// TIA Portal V19 export
FUNCTION "Route 405" : Void   // FC104, STL
TITLE = Polygon Transfer Line - SIP Sequence
{ S7_Optimized_Access := 'TRUE' }
// stored: AutoNumber false
   VAR_TEMP
      device_fault : Bool;
      switch_fault : Bool;
      tmp : Bool;
      Step_on : Bool;
      Dev_Check : Bool;
      New_Msg : Bool;
      Route_Ready : Bool;   // Ready to Run
      PNIOnodeFault : Bool;
      StepTime : S5Time;
      TimerError : Int;
      scratch_DI : DInt;
      scratch_Real : Real;
      Message : Int;
      scratch_I : Int;
      tmpWord : Word;
      PNIODiag : Struct
         node_2 : Struct
            failed : Bool;
            moduleFault : Bool;
         END_STRUCT;
         node_3 : Struct
            failed : Bool;
            moduleFault : Bool;
         END_STRUCT;
         node_4 : Struct
            failed : Bool;
            moduleFault : Bool;
         END_STRUCT;
         node_5 : Struct
            failed : Bool;
            moduleFault : Bool;
         END_STRUCT;
         node_6 : Struct
            failed : Bool;
            moduleFault : Bool;
         END_STRUCT;
         node_7 : Struct
            failed : Bool;
            moduleFault : Bool;
         END_STRUCT;
         node_8 : Struct
            failed : Bool;
            moduleFault : Bool;
         END_STRUCT;
         node_9 : Struct
            failed : Bool;
            moduleFault : Bool;
         END_STRUCT;
         node_10 : Struct
            failed : Bool;
            moduleFault : Bool;
         END_STRUCT;
         node_11 : Struct
            failed : Bool;
            moduleFault : Bool;
         END_STRUCT;
         node_12 : Struct
            failed : Bool;
            moduleFault : Bool;
         END_STRUCT;
      END_STRUCT;
      __PlcmigTempFillBits_38B0 : Array[0..7] of Bool;
   END_VAR
BEGIN

NETWORK
TITLE = PNIO 100 Node Faults
// PNIO Node 2
// PNIO Node 2
      A     "Module Diagnostic Result"."2_AL1103".ErrorValue.%X1;
      =     #PNIODiag.node_2.failed;
      A     "Module Diagnostic Result"."2_AL1103".ErrorValue.%X2;
      =     #PNIODiag.node_2.moduleFault;
// PNIO Node 3
      A     "Module Diagnostic Result"."3_AL1307".ErrorValue.%X1;
      =     #PNIODiag.node_3.failed;
      A     "Module Diagnostic Result"."3_AL1307".ErrorValue.%X2;
      =     #PNIODiag.node_3.moduleFault;
// PNIO Node 4
      A     "Module Diagnostic Result"."4_AL1307".ErrorValue.%X1;
      =     #PNIODiag.node_4.failed;
      A     "Module Diagnostic Result"."4_AL1307".ErrorValue.%X2;
      =     #PNIODiag.node_4.moduleFault;
// PNIO Node 5
      A     "Module Diagnostic Result"."5_AL1307".ErrorValue.%X1;
      =     #PNIODiag.node_5.failed;
      A     "Module Diagnostic Result"."5_AL1307".ErrorValue.%X2;
      =     #PNIODiag.node_5.moduleFault;
// PNIO Node 6
      A     "Module Diagnostic Result"."6_AL1307".ErrorValue.%X1;
      =     #PNIODiag.node_6.failed;
      A     "Module Diagnostic Result"."6_AL1307".ErrorValue.%X2;
      =     #PNIODiag.node_6.moduleFault;
// PNIO Node 7
      A     "Module Diagnostic Result"."7_AL1307".ErrorValue.%X1;
      =     #PNIODiag.node_7.failed;
      A     "Module Diagnostic Result"."7_AL1307".ErrorValue.%X2;
      =     #PNIODiag.node_7.moduleFault;
// PNIO Node 8
      A     "Module Diagnostic Result"."8_Promag300".ErrorValue.%X1;
      =     #PNIODiag.node_8.failed;
      A     "Module Diagnostic Result"."8_Promag300".ErrorValue.%X2;
      =     #PNIODiag.node_8.moduleFault;
// PNIO Node 9
      A     "Module Diagnostic Result"."9_SinaG120".ErrorValue.%X1;
      =     #PNIODiag.node_9.failed;
      A     "Module Diagnostic Result"."9_SinaG120".ErrorValue.%X2;
      =     #PNIODiag.node_9.moduleFault;
// PNIO Node 10
      A     "Module Diagnostic Result"."10_AL1307".ErrorValue.%X1;
      =     #PNIODiag.node_10.failed;
      A     "Module Diagnostic Result"."10_AL1307".ErrorValue.%X2;
      =     #PNIODiag.node_10.moduleFault;
// PNIO Node 11
      A     "Module Diagnostic Result"."11_PNCoup".ErrorValue.%X1;
      =     #PNIODiag.node_11.failed;
      A     "Module Diagnostic Result"."11_PNCoup".ErrorValue.%X2;
      =     #PNIODiag.node_11.moduleFault;
// PNIO Node 12
      A     "Module Diagnostic Result"."12_AL1307".ErrorValue.%X1;
      =     #PNIODiag.node_12.failed;
      A     "Module Diagnostic Result"."12_AL1307".ErrorValue.%X2;
      =     #PNIODiag.node_12.moduleFault;


NETWORK
TITLE = PNIO node fault
      O     #PNIODiag.node_2.failed;
      O     #PNIODiag.node_2.moduleFault;
      O     #PNIODiag.node_3.failed;
      O     #PNIODiag.node_3.moduleFault;
      O     #PNIODiag.node_4.failed;
      O     #PNIODiag.node_4.moduleFault;
      O     #PNIODiag.node_5.failed;
      O     #PNIODiag.node_5.moduleFault;
      O     #PNIODiag.node_6.failed;
      O     #PNIODiag.node_6.moduleFault;
      O     #PNIODiag.node_7.failed;
      O     #PNIODiag.node_7.moduleFault;
      O     #PNIODiag.node_8.failed;
      O     #PNIODiag.node_8.moduleFault;
      O     #PNIODiag.node_9.failed;
      O     #PNIODiag.node_9.moduleFault;
      O     #PNIODiag.node_10.failed;
      O     #PNIODiag.node_10.moduleFault;
      O     #PNIODiag.node_11.failed;
      O     #PNIODiag.node_11.moduleFault;
      O     #PNIODiag.node_12.failed;
      O     #PNIODiag.node_12.moduleFault;
      =     #PNIOnodeFault;


NETWORK
TITLE = Device Faults
      O     "ItemAlarmsOP".Item[20];  //FB_FAULT_VALVE_09_05
      O     "ItemAlarmsOP".Item[23];  //FB_FAULT_VALVE_09_08
      O     "ItemAlarmsOP".Item[24];  //FB_FAULT_VALVE_09_09
      O     "ItemAlarmsOP".Item[25];  //FB_FAULT_VALVE_09_10
      O     "ItemAlarmsOP".Item[26];  //FB_FAULT_VALVE_09_11
      O     "ItemInfoScada".Items[68].fb_error;
      O     "ItemInfoScada".Items[69].fb_error;
      O     "ItemInfoScada".Items[70].fb_error;
      O     "ItemInfoScada".Items[85].fb_error;
      O     "ItemInfoScada".Items[71].fb_error;
      O     "ItemInfoScada".Items[72].fb_error;
      O     "ItemInfoScada".Items[73].fb_error;
      O     "ItemInfoScada".Items[74].fb_error;
      O     "ItemInfoScada".Items[75].fb_error;
      O     "ItemInfoScada".Items[76].fb_error;
      O     "ItemInfoScada".Items[78].fb_error;
      O     "ItemInfoScada".Items[79].fb_error;
      O     "ItemInfoScada".Items[80].fb_error;
      O     "ItemInfoScada".Items[81].fb_error;
      O     "ItemInfoScada".Items[82].fb_error;
      O     "ItemInfoScada".Items[83].fb_error;
      O     "ItemInfoScada".Items[77].fb_error;
      O     "ItemInfoScada".Items[84].fb_error;
      O     "ItemInfoScada".Items[77].TrippedInd;
      O     "ItemInfoScada".Items[77].IsolatedInd;
      O     "ItemInfoScada".Items[84].TrippedInd;
      O     "ItemInfoScada".Items[84].IsolatedInd;
      O     #PNIOnodeFault;
      O     "ProcessAndPbAlarms"."A"[78];  //A78_PG_PTX0940HighPress
      AN    "RTE_405_TestBit";
      =     #device_fault;

NETWORK
TITLE = Switch Fault
      A(;
      ON    "PG_Devices".DI_100_005_X06_X1_3p4;
      O     "PG_Devices".DI_100_005_X06_X1_3p2;
      O     "PG_Devices".DI_100_012_X1_1p2;
      );
      AN    "RTE_405_TestBit";
      =     #switch_fault;

NETWORK
TITLE = Set Devices in Auto
      A     "RTE_405_DB".HMI.RUNNING;
      R     "ItemInfoScada".Items[50].auto_man;
      R     "ItemInfoScada".Items[53].auto_man;
      R     "ItemInfoScada".Items[54].auto_man;
      R     "ItemInfoScada".Items[55].auto_man;
      R     "ItemInfoScada".Items[56].auto_man;
      R     "ItemInfoScada".Items[69].auto_man;
      R     "ItemInfoScada".Items[70].auto_man;
      R     "ItemInfoScada".Items[68].auto_man;
      R     "ItemInfoScada".Items[72].auto_man;
      R     "ItemInfoScada".Items[73].auto_man;
      R     "ItemInfoScada".Items[75].auto_man;
      R     "ItemInfoScada".Items[76].auto_man;
      R     "ItemInfoScada".Items[78].auto_man;
      R     "ItemInfoScada".Items[79].auto_man;
      R     "ItemInfoScada".Items[80].auto_man;
      R     "ItemInfoScada".Items[81].auto_man;
      R     "ItemInfoScada".Items[82].auto_man;
      R     "ItemInfoScada".Items[83].auto_man;
      R     "ItemInfoScada".Items[77].auto_man;
      R     "ItemInfoScada".Items[84].auto_man;

NETWORK
TITLE = Route Healthy
      AN    #device_fault;
      AN    #switch_fault;
      =     "RTE_405_DB".HMI.Route_Healthy;

NETWORK
TITLE = DEVICE FAULT STATUS
      A     #device_fault;
      =     "RTE_405_DB".FLAGS.Device_Fault;

NETWORK
TITLE = GENERAL FAULT STATUS
      O     #switch_fault;
      O     "RTE_405_DB".FLAGS.Device_Fault;
      A     "RTE_405_DB".HMI.RUNNING;
      =     "RTE_405_DB".HMI.FAULT;

NETWORK
TITLE = Temporary Message Store
// Clear down temporary message store.
      L     0;
      T     #Message;
      NOP   0;

NETWORK
TITLE = Generate Sequence Start Command
// The sequence is initiated via the interface signals ..afl
      A     "RTE_405_DB".HMI_CMD.Start;
      AN    "RTE_405_DB".HMI.RUNNING;
      A     "RTE_405_DB".HMI.Route_Healthy;
      =     "RTE_405_DB".FLAGS.Sequence_Start;

      AN    "RTE_405_DB".HMI.RUNNING;
      A     "RTE_405_DB".HMI.Route_Healthy;
      =     "RTE_405_DB".HMI_CMD.Start_Available;


NETWORK
TITLE = ****ERROR MESSAGE****
// Message 10 - Device Fault
      A(;
      O     "RTE_405_DB".HMI_CMD.Start;
      O     "RTE_405_DB".HMI_CMD.Continue;
      );
      A     #device_fault;
      JNB   _001;
      L     10;
      T     #Message;
      SET;
      SAVE;
      CLR;
_001: A     BR;
      JC    AA01;

NETWORK
TITLE = ****ERROR MESSAGE****
// Message 12 - Forward Control stop activated
      A(;
      O     "RTE_405_DB".HMI_CMD.Start;
      O     "RTE_405_DB".HMI_CMD.Continue;
      );
      A     "PG_Devices".DI_100_012_X1_1p2;
      JNB   _002;
      L     12;
      T     #Message;
      SET;
      SAVE;
      CLR;
_002: A     BR;
      JC    AA01;

NETWORK
TITLE = ****ERROR MESSAGE****
// Message 37 - Swingbend out of position
      A(;
      O     "RTE_405_DB".HMI_CMD.Start;
      O     "RTE_405_DB".HMI_CMD.Continue;
      );
      A(;
      O     "PG_Devices".DI_100_005_X06_X1_3p2;
      ON    "PG_Devices".DI_100_005_X06_X1_3p4;
      );
      JNB   _003;
      L     37;
      T     #Message;
      SET;
      SAVE;
      CLR;
_003: A     BR;
      JC    AA01;

NETWORK
TITLE = ****ERROR MESSAGE****
// Message 17 - Sequence Not Held
// To abort or continue the clean it must have already been held.
      A(;
      O     "RTE_405_DB".HMI_CMD.Abort;
      O     "RTE_405_DB".HMI_CMD.Continue;
      );
      AN    "RTE_405_DB".HMI.SEQUENCE_HELD;
      JNB   _004;
      L     17;
      T     #Message;
      SET;
      SAVE;
      CLR;
_004: A     BR;
      JC    AA01;

NETWORK
TITLE = ****ERROR MESSAGE****
// Message 57 - Line not clean
      A(;
      O     "RTE_405_DB".HMI_CMD.Start;
      O     "RTE_405_DB".HMI_CMD.Continue;
      );
      AN    "RTE_404_DB".FLAGS.Clean;
      JNB   _005;
      L     57;
      T     #Message;
      SET;
      SAVE;
      CLR;
_005: A     BR;
      JC    AA01;

NETWORK
TITLE = ****ERROR MESSAGE****
// Message 21 - Tank not sterilising or sterile
      AN    "RTE_405_DB".FLAGS.Sterile;
      A(;
      O     "RTE_405_DB".HMI_CMD.Start;
      O     "RTE_405_DB".HMI_CMD.Continue;
      );
      AN    "S0 PRESTERILIZING";
      AN    "TANK STERILE";
      JNB   _006;
      L     21;
      T     #Message;
      SET;
      SAVE;
      CLR;
_006: A     BR;
      JC    AA01;

NETWORK
TITLE = ****ERROR MESSAGE****
// Message 22 - Line In Production
// *** Use Production Seq running bit ***
      A(;
      O     "RTE_405_DB".HMI_CMD.Start;
      O     "RTE_405_DB".HMI_CMD.Continue;
      );
      A     "RTE_406_DB".HMI.RUNNING;
      JNB   _007;
      L     22;
      T     #Message;
      SET;
      SAVE;
      CLR;
_007: A     BR;
      JC    AA01;

NETWORK
TITLE = New Message Detected
AA01: A(;
      L     #Message;
      L     0;
      <>I;
      );
      JNB   _008;
      L     #Message;
      T     "RTE_405_DB".HMI.ERROR_TEXT_NUMBER;
      SET;
      SAVE;
      CLR;
_008: A     BR;
      =     #New_Msg;

NETWORK
TITLE = ****NEW ERROR MESSAGE****
// Reset all CIP commands except START.
// On a new non-zero error message being displayed reset all commands from SCADA 
// so they take no action. Also, start a delay off timer to cancel display of the 
// error message.
      A     #New_Msg;
      R     "RTE_405_DB".HMI_CMD.Abort;
      R     "RTE_405_DB".HMI_CMD.Continue;
      R     "RTE_405_DB".HMI_CMD.Hold;
      R     "RTE_405_DB".HMI_CMD.Timer_Release;
      R     "RTE_405_DB".HMI_CMD.Timer_Hold;
      R     "RTE_405_DB".FLAGS.Sequence_Start;
      L     S5T#10S;
      SF    "RTE405_MSG";

NETWORK
TITLE = ****NEW ERROR MESSAGE****
// Error message display cancel.
      AN    "RTE405_MSG";
      JNB   _009;
      L     0;
      T     "RTE_405_DB".HMI.ERROR_TEXT_NUMBER;
_009: NOP   0;

NETWORK
TITLE = ROUTE RUNNING
      L     "RTE_405_DB".HMI.STEP_NUMBER;
      L     0;
      <>I;
      =     "RTE_405_DB".HMI.RUNNING;

NETWORK
TITLE = ****SEQ ABORT****
      A(;
      O     "RTE_405_DB".HMI_CMD.Abort;
      O;
      AN    "S0 PRESTERILIZING";
      AN    "TANK STERILE";
      O     "ProcessAndPbAlarms"."A"[77];  //A77_PG_SIP_HighHighTemp
      );
      A     "RTE_405_DB".HMI.SEQUENCE_HELD;
      S     "RTE_405_DB".HMI.SEQUENCE_ABORTED;

      A     "RTE_405_DB".HMI.SEQUENCE_HELD;
      =     "RTE_405_DB".HMI_CMD.Abort_Available;


NETWORK
TITLE = Enable HMI Hold Pb
      A     "RTE_405_DB".HMI.RUNNING;
      =     "RTE_405_DB".HMI_CMD.Hold_Available;

NETWORK
TITLE = Sequence held flag
// Set sequence hold if sequence is running and a hold fault condition is detected 
// or a sequence hold command is received from SCADA.
// 
// When a validated CONTINUE command is received from SCADA and all fault 
// conditions are cleared then reset sequence hold.
// 
// Added "seq Aborted" if not Step0 to Reset "seq Held" if seq is auto aborted if 
// running and Tank not sterilising or Sterile.
      A(;
      O     "RTE_405_DB".HMI_CMD.Hold;
      ON    "RTE_405_DB".HMI.Route_Healthy;
      O;
      AN    "S0 PRESTERILIZING";
      AN    "TANK STERILE";
      O     "ProcessAndPbAlarms"."A"[77];  //A77_PG_SIP_HighHighTemp
      );
      A     "RTE_405_DB".HMI.RUNNING;
      =     #__PlcmigTempFillBits_38B0[0];
      A     #__PlcmigTempFillBits_38B0[0];
      BLD   102;
      S     "RTE_405_DB".HMI.SEQUENCE_HELD;
      A     #__PlcmigTempFillBits_38B0[0];
      NOT;
      =     #__PlcmigTempFillBits_38B0[1];
      A     #__PlcmigTempFillBits_38B0[1];
      A(;
      O     "RTE_405_DB".HMI_CMD.Continue;
      O     "RTE_405_DB".HMI_CMD.Abort;
      O;
      A     "RTE_405_DB".HMI.SEQUENCE_ABORTED;
      AN    "RTE_405_DB".FLAGS.STEP_0;
      );
      R     "RTE_405_DB".HMI.SEQUENCE_HELD;
      A     #__PlcmigTempFillBits_38B0[1];
      A     "RTE_405_DB".HMI.SEQUENCE_HELD;
      =     "RTE_405_DB".HMI_CMD.Continue_Available;

NETWORK
TITLE = Sequence held flag
// Reset when circuit not running i.e after an abort.
      A     "RTE_405_DB".FLAGS.STEP_0;
      AN    "RTE_405_DB".HMI.RUNNING;
      R     "RTE_405_DB".HMI.SEQUENCE_HELD;

NETWORK
TITLE = ****RESET ABORT FLAG****
      A     "RTE_405_DB".FLAGS.STEP_0;
      A     "RTE_405_DB".FLAGS.Step_Change;
      R     "RTE_405_DB".HMI.SEQUENCE_ABORTED;

NETWORK
TITLE = Step 0.0 Reset
      AN    "RTE_405_DB".HMI.RUNNING;
      AN    "RTE_405_DB".FLAGS.STEP_0;
      =     #Step_on;

NETWORK
TITLE = Step 0.0 Reset
// Reset sequnece to step 0 and clear down step value and dimension words.
      A(;
      A(;
      A(;
      O     #Step_on;
      O;
      A     "RTE_405_DB".FLAGS.STEP_0;
      A     "RTE_405_DB".FLAGS.Step_Change;
      );
      JNB   _00a;
      L     0;
      T     "RTE_405_DB".HMI.NEXT_STEP;
      SET;
      SAVE;
      CLR;
_00a: A     BR;
      );
      JNB   _00b;
      L     0;
      T     "RTE_405_DB".HMI.STEP_VALUE;
      SET;
      SAVE;
      CLR;
_00b: A     BR;
      );
      JNB   _00c;
      L     0;
      T     "RTE_405_DB".HMI.STEP_VALUE_DIMENSION;
_00c: NOP   0;

NETWORK
TITLE = Move to Step 1.0
      A     "RTE_405_DB".FLAGS.STEP_0;
      A     "RTE_405_DB".FLAGS.Sequence_Start;
      A     "RTE_404_DB".FLAGS.Clean;
      A(;
      O     "S0 PRESTERILIZING";
      O     "TANK STERILE";
      );
      =     #__PlcmigTempFillBits_38B0[0];
      A     #__PlcmigTempFillBits_38B0[0];
      BLD   102;
      =     #Step_on;
      A     #__PlcmigTempFillBits_38B0[0];
      JNB   _00d;
      L     10;
      T     "RTE_405_DB".HMI.NEXT_STEP;
_00d: NOP   0;

NETWORK
TITLE = Move to Step 2.0 - Dev Check
// Dev Check following Route valves Open - 09.10, 09.08, 09.45, 10.21, 10.23, 10.25
// and following Route Valves closed - 09.09, 09.05, 10.24
      A     "RTE_405_DB".FLAGS.STEP_1_0;
      A     "Y0903";
      A     "Y0905R";
      A     "Y0908S";
      A     "Y0909S";
      A     "Y0910R";
      A     "Y0911R";
      A     "ItemInfoScada".Items[68].Set_FB;
      A     "ItemInfoScada".Items[69].Set_FB;
      A     "ItemInfoScada".Items[70].Reset_FB;
      =     #Dev_Check;

NETWORK
TITLE = Move to Step 2.0 - Dev Check
      A     #Dev_Check;
      A     "ItemInfoScada".Items[71].Reset_FB;
      A     "ItemInfoScada".Items[72].Set_FB;
      A     "ItemInfoScada".Items[73].Set_FB;
      A     "ItemInfoScada".Items[75].Set_FB;
      A     "ItemInfoScada".Items[76].Set_FB;
      A     "ItemInfoScada".Items[78].Set_FB;
      A     "ItemInfoScada".Items[79].Reset_FB;
      A     "ItemInfoScada".Items[80].Reset_FB;
      =     #Dev_Check;

NETWORK
TITLE = Move to Step 2.0 - Dev Check
      A     #Dev_Check;
      A     "ItemInfoScada".Items[81].Reset_FB;
//   A     "ItemInfoScada".items[82].Set_FB
//    A     "ItemInfoScada".items[83].Set_FB
      A     "ItemInfoScada".Items[77].Reset_FB;
      A     "ItemInfoScada".Items[84].Set_FB;
      =     #Dev_Check;

NETWORK
TITLE = Move to Step 2.0
      A     "RTE_405_DB".FLAGS.STEP_1_0;
      A     #Dev_Check;
      AN    "RTE_405_DB".FLAGS.Step_Change;
      =     #__PlcmigTempFillBits_38B0[0];
      A     #__PlcmigTempFillBits_38B0[0];
      BLD   102;
      =     #Step_on;
      A     #__PlcmigTempFillBits_38B0[0];
      JNB   _00e;
      L     20;
      T     "RTE_405_DB".HMI.NEXT_STEP;
_00e: NOP   0;

NETWORK
TITLE = Move to Step 3.0 - Temperature Check
      A     "RTE_405_DB".FLAGS.STEP_2_0;
      A(;
      L     "PG_Devices".TTX1040.Value;  // PG EOL
      L     130.0;
      >=R;
      );
      A(;
      L     "PG_Devices".TTX1041.Value;  //  PG EOL
      L     130.0;
      >=R;
      );
      A(;
      L     "PG_Devices".TTX0940.Value;  // AHV - Transfer line - Sterile Air Barrier
      L     130.0;
      >=R;
      );
      A(;
      L     "PG_Devices".TTX0941.Value;  // M0940 Condensate
      L     130.0;
      >=R;
      );
      =     #tmp;

NETWORK
TITLE = Move to Step 3.0
      A     "RTE_405_DB".FLAGS.STEP_2_0;
      A(;
      L     "MeasuredValues".TT0950REAL;
      L     130.0;
      >=R;
      );
      A     #tmp;
      AN    "RTE_405_DB".FLAGS.Step_Change;
      =     #__PlcmigTempFillBits_38B0[0];
      A     #__PlcmigTempFillBits_38B0[0];
      BLD   102;
      =     #Step_on;
      A     #__PlcmigTempFillBits_38B0[0];
      JNB   _00f;
      L     30;
      T     "RTE_405_DB".HMI.NEXT_STEP;
_00f: NOP   0;

NETWORK
TITLE = Initialise Step Parameters
      A(;
      A     #Step_on;
      JNB   _010;
      L     "RTE_405_DB".PARAMETERS.PARAM_01;
      T     "RTE_405_DB".HMI.STEP_VALUE;
      SET;
      SAVE;
      CLR;
_010: A     BR;
      );
      JNB   _011;
      L     1;
      T     "RTE_405_DB".HMI.STEP_VALUE_DIMENSION;
_011: NOP   0;

NETWORK
TITLE = Move to Step 4.0
      A     "RTE_405_DB".FLAGS.STEP_3_0;
      A(;
      O     "TANK STERILE";
      O     "m19.3";
      );
      A     "RTE_405_DB".FLAGS.Step_Value_Done;
      AN    "RTE_405_DB".FLAGS.Step_Change;
      =     #__PlcmigTempFillBits_38B0[0];
      A     #__PlcmigTempFillBits_38B0[0];
      BLD   102;
      =     #Step_on;
      A     #__PlcmigTempFillBits_38B0[0];
      JNB   _012;
      L     40;
      T     "RTE_405_DB".HMI.NEXT_STEP;
_012: NOP   0;

NETWORK
TITLE = Move back to Step 2.0
      A     "RTE_405_DB".FLAGS.STEP_3_0;
      A(;
      O(;
      L     "PG_Devices".TTX1040.Value;
      L     123.0;
      <R;
      );
      O(;
      L     "PG_Devices".TTX1041.Value;
      L     123.0;
      <R;
      );
      O(;
      L     "PG_Devices".TTX0940.Value;
      L     123.0;
      <R;
      );
      O(;
      L     "PG_Devices".TTX0941.Value;
      L     123.0;
      <R;
      );
      O(;
      L     "MeasuredValues".TT0950REAL;
      L     123.0;
      <R;
      );
      );
      AN    "RTE_405_DB".FLAGS.Step_Change;
      =     #__PlcmigTempFillBits_38B0[0];
      A     #__PlcmigTempFillBits_38B0[0];
      BLD   102;
      =     #Step_on;
      A     #__PlcmigTempFillBits_38B0[0];
      JNB   _013;
      L     20;
      T     "RTE_405_DB".HMI.NEXT_STEP;
_013: NOP   0;
      A     #__PlcmigTempFillBits_38B0[0];
      JNB   _014;
      L     0;
      T     "RTE_405_DB".HMI.STEP_VALUE;
_014: NOP   0;

NETWORK
TITLE = Device Check
      A     "RTE_405_DB".FLAGS.STEP_4_0;
      A     "ItemInfoScada".Items[69].Set_FB;
      A     "ItemInfoScada".Items[70].Set_FB;
      A     "ItemInfoScada".Items[71].Set_FB;
      A     "ItemInfoScada".Items[73].Set_FB;
      A     "ItemInfoScada".Items[75].Set_FB;
      A     "ItemInfoScada".Items[78].Set_FB;
      A     "ItemInfoScada".Items[79].Reset_FB;
      A     "ItemInfoScada".Items[68].Reset_FB;
      A     "ItemInfoScada".Items[76].Reset_FB;
      =     #Dev_Check;

NETWORK
TITLE = Move to Step 5.0
      A     "RTE_405_DB".FLAGS.STEP_4_0;
      A     #Dev_Check;
      AN    "RTE_405_DB".FLAGS.Step_Change;
      =     #__PlcmigTempFillBits_38B0[0];
      A     #__PlcmigTempFillBits_38B0[0];
      BLD   102;
      =     #Step_on;
      A     #__PlcmigTempFillBits_38B0[0];
      JNB   _015;
      L     50;
      T     "RTE_405_DB".HMI.NEXT_STEP;
_015: NOP   0;

NETWORK
TITLE = Move to Step 6.0
      A     "RTE_405_DB".FLAGS.STEP_5_0;
      A(;
      L     "PG_Devices".TTX0942.Value;
      L     40.0;
      <R;
      );
      AN    "RTE_405_DB".FLAGS.Step_Change;
      =     #__PlcmigTempFillBits_38B0[0];
      A     #__PlcmigTempFillBits_38B0[0];
      BLD   102;
      =     #Step_on;
      A     #__PlcmigTempFillBits_38B0[0];
      JNB   _016;
      L     60;
      T     "RTE_405_DB".HMI.NEXT_STEP;
_016: NOP   0;

NETWORK
TITLE = Dev Check
// Check following valve V10.24 are open, and v09.08, v09.10, V10.24 are shut
      A     "RTE_405_DB".FLAGS.STEP_6_0;
      A     "Y0908R";
      A     "Y0910R";
      A     "ItemInfoScada".Items[78].Reset_FB;
      A     "ItemInfoScada".Items[80].Set_FB;
      =     #Dev_Check;

NETWORK
TITLE = Move to Step 7.0
// Need to start monitoring TT1020, TT1040, and TT1041
      A     "RTE_405_DB".FLAGS.STEP_6_0;
      A     #Dev_Check;
      AN    "RTE_405_DB".FLAGS.Step_Change;
      =     #__PlcmigTempFillBits_38B0[0];
      A     #__PlcmigTempFillBits_38B0[0];
      BLD   102;
      =     #Step_on;
      A     #__PlcmigTempFillBits_38B0[0];
      JNB   _017;
      L     70;
      T     "RTE_405_DB".HMI.NEXT_STEP;
_017: NOP   0;

NETWORK
TITLE = Dev Check
// Check following valve are closed  V09.40, V09.42, V09.44
      A     "RTE_405_DB".FLAGS.STEP_7_0;
      A     "ItemInfoScada".Items[71].Reset_FB;
      A     "ItemInfoScada".Items[72].Set_FB;
      A     "ItemInfoScada".Items[73].Reset_FB;
      A     "ItemInfoScada".Items[74].Set_FB;
      A     "ItemInfoScada".Items[75].Reset_FB;
      A     "Y0902";
      =     #Dev_Check;

NETWORK
TITLE = Move to Step 8.0
// In step 8 need to start monitoring TT0940
      A     "RTE_405_DB".FLAGS.STEP_7_0;
      A     #Dev_Check;
      AN    "RTE_405_DB".FLAGS.Step_Change;
      =     #__PlcmigTempFillBits_38B0[0];
      A     #__PlcmigTempFillBits_38B0[0];
      BLD   102;
      =     #Step_on;
      A     #__PlcmigTempFillBits_38B0[0];
      JNB   _018;
      L     80;
      T     "RTE_405_DB".HMI.NEXT_STEP;
_018: NOP   0;

NETWORK
TITLE = Set Polygon Transfer Line Sterile Status
// Check following valve are closed  V09.40, V09.42, V09.44
      A     "RTE_405_DB".FLAGS.STEP_8_0;
      S     "RTE_405_DB".FLAGS.Sterile;
      A(;
      A     "RTE_405_DB".FLAGS.STEP_0;
      A     "RTE_405_DB".FLAGS.Sequence_Start;
      O;
      A     "AFI";
      AN    "TANK STERILE";
      A     "RTE_405_DB".FLAGS.Sterile;
      );
      R     "RTE_405_DB".FLAGS.Sterile;
      NOP   0;

NETWORK
TITLE = Move to Step 9.0 - END
      A     "RTE_405_DB".FLAGS.STEP_8_0;
      A     "RTE_405_DB".FLAGS.Sterile;
      A(;
      O     "RTE_405_DB".FLAGS.Production_Req;
      O     "RTE_405_DB".FLAGS.Sterile;
      );
      AN    "RTE_405_DB".FLAGS.Step_Change;
      =     #__PlcmigTempFillBits_38B0[0];
      A     #__PlcmigTempFillBits_38B0[0];
      BLD   102;
      =     #Step_on;
      A     #__PlcmigTempFillBits_38B0[0];
      JNB   _019;
      L     90;
      T     "RTE_405_DB".HMI.NEXT_STEP;
_019: NOP   0;

NETWORK
TITLE = Move to Step 0.0
      A(;
      A     "RTE_405_DB".FLAGS.STEP_END;
      A     "RTE_405_DB".FLAGS.Step_Value_Done;
      O     "RTE_405_DB".HMI.SEQUENCE_ABORTED;
      );
      AN    "RTE_405_DB".FLAGS.Step_Change;
      =     #__PlcmigTempFillBits_38B0[0];
      A     #__PlcmigTempFillBits_38B0[0];
      BLD   102;
      =     #Step_on;
      A     #__PlcmigTempFillBits_38B0[0];
      JNB   _01a;
      L     0;
      T     "RTE_405_DB".HMI.NEXT_STEP;
_01a: NOP   0;

NETWORK
TITLE = Step Change Detected
// The next step number is different to the current step then set flag.
      L     "RTE_405_DB".HMI.NEXT_STEP;
      L     "RTE_405_DB".HMI.STEP_NUMBER;
      <>I;
      =     "RTE_405_DB".FLAGS.Step_Change;

NETWORK
TITLE = Current step value decremented to zero
      A(;
      L     "RTE_405_DB".HMI.STEP_VALUE;
      L     0;
      <=I;
      );
      AN    "RTE_405_DB".FLAGS.Step_Change;
      =     "RTE_405_DB".FLAGS.Step_Value_Done;

NETWORK
TITLE = Enable step count down
      A(;
      A     "RTE_405_DB".FLAGS.STEP_3_0;
      A(;
      O(;
      L     "PG_Devices".TTX1040.Value;
      L     130.0;
      <R;
      );
      O(;
      L     "PG_Devices".TTX1041.Value;
      L     130.0;
      <R;
      );
      O(;
      L     "PG_Devices".TTX0940.Value;
      L     130.0;
      <R;
      );
      O(;
      L     "PG_Devices".TTX0941.Value;
      L     130.0;
      <R;
      );
      O(;
      L     "MeasuredValues".TT0950REAL;
      L     130.0;
      <R;
      );
      );
      O     "RTE_405_DB".HMI.SEQUENCE_HELD;
      );
      NOT;
      =     "RTE_405_DB".FLAGS.Step_Count_Enable;

NETWORK
TITLE = Decrement Step Value
// With count enabled and timer not held count down on each 1 second pulse.
      A     "RTE_405_DB".HMI.RUNNING;
      A     "RTE_405_DB".FLAGS.Step_Count_Enable;
      AN    "RTE_405_DB".HMI.TIMER_HELD;
      AN    "RTE_405_DB".FLAGS.Step_Value_Done;
      A     "1HZ_ONESHOT";
      JNB   _01b;
      L     "RTE_405_DB".HMI.STEP_VALUE;
      L     1;
      -I;
      T     "RTE_405_DB".HMI.STEP_VALUE;
_01b: NOP   0;

NETWORK
TITLE = Reset HMI commands
      A     "ATI";
      R     "RTE_405_DB".HMI_CMD.Abort;
      R     "RTE_405_DB".HMI_CMD.Continue;
      R     "RTE_405_DB".HMI_CMD.Hold;
      R     "RTE_405_DB".HMI_CMD.Timer_Release;
      R     "RTE_405_DB".HMI_CMD.Timer_Hold;
      R     "RTE_405_DB".HMI_CMD.Start;

NETWORK
TITLE = MESSAGE CLEARANCE TIMING
      A     "1HZ_ONESHOT";
      =     #__PlcmigTempFillBits_38B0[0];
      BLD   103;
      CALL  "ERROR_MSG_CLEAR"
      ( MESSAGE_CLEAR_TIME := 10,
        SECOND_PULSE       := #__PlcmigTempFillBits_38B0[0],
        ERROR_MESSAGE      := "RTE_405_DB".HMI.ERROR_TEXT_NUMBER,
        ERROR_MESSAGE_MEM  := "RTE_405_DB".CONTROL.ERROR_MESSAGE_MEM,
        ELAPSED_TIME       := "RTE_405_DB".CONTROL.MESSAGE_TIME
      );
      NOP   0;

NETWORK
TITLE = STEP TIMER
// On detection of a new step, the timer is reset to 0 and will then start timing 
// whilst on the current step.
      A     "1HZ_ONESHOT";
      =     #__PlcmigTempFillBits_38B0[0];
      BLD   103;
      CALL  "STEP_TIMER"
      ( DBNR                   := 405,
        NEXT_STEP_LOCATION     := 18,
        STEP_NUM_LOCATION      := 2,
        TIME_PULSE             := #__PlcmigTempFillBits_38B0[0],
        STEP_TIME_ACC_LOCATION := 26
      );
      NOP   0;

NETWORK
TITLE = 
      A     "RTE_405_DB".FLAGS.Step_Change;
      JNB   _01c;
      L     "RTE_405_DB".HMI.NEXT_STEP;
      T     "RTE_405_DB".HMI.STEP_NUMBER;
_01c: NOP   0;

NETWORK
TITLE = Spare
      L     "RTE_405_DB".HMI.STEP_NUMBER;
      L     0;
      ==I;
      =     "RTE_405_DB".FLAGS.STEP_0;

NETWORK
TITLE = Spare
      O     "RTE_405_DB".HMI.RUNNING;
      ON    "RTE_405_DB".HMI.RUNNING;
      =     #__PlcmigTempFillBits_38B0[0];
      A     #__PlcmigTempFillBits_38B0[0];
      A(;
      L     "RTE_405_DB".HMI.STEP_NUMBER;
      L     10;
      ==I;
      );
      =     "RTE_405_DB".FLAGS.STEP_1_0;
      A     #__PlcmigTempFillBits_38B0[0];
      A(;
      L     "RTE_405_DB".HMI.STEP_NUMBER;
      L     20;
      ==I;
      );
      =     "RTE_405_DB".FLAGS.STEP_2_0;
      A     #__PlcmigTempFillBits_38B0[0];
      A(;
      L     "RTE_405_DB".HMI.STEP_NUMBER;
      L     30;
      ==I;
      );
      =     "RTE_405_DB".FLAGS.STEP_3_0;
      A     #__PlcmigTempFillBits_38B0[0];
      A(;
      L     "RTE_405_DB".HMI.STEP_NUMBER;
      L     40;
      ==I;
      );
      =     "RTE_405_DB".FLAGS.STEP_4_0;
      A     #__PlcmigTempFillBits_38B0[0];
      A(;
      L     "RTE_405_DB".HMI.STEP_NUMBER;
      L     50;
      ==I;
      );
      =     "RTE_405_DB".FLAGS.STEP_5_0;
      A     #__PlcmigTempFillBits_38B0[0];
      A(;
      L     "RTE_405_DB".HMI.STEP_NUMBER;
      L     60;
      ==I;
      );
      =     "RTE_405_DB".FLAGS.STEP_6_0;
      A     #__PlcmigTempFillBits_38B0[0];
      A(;
      L     "RTE_405_DB".HMI.STEP_NUMBER;
      L     70;
      >=I;
      );
      =     "RTE_405_DB".FLAGS.STEP_7_0;
      A     #__PlcmigTempFillBits_38B0[0];
      A(;
      L     "RTE_405_DB".HMI.STEP_NUMBER;
      L     80;
      >=I;
      );
      =     "RTE_405_DB".FLAGS.STEP_8_0;
      A     #__PlcmigTempFillBits_38B0[0];
      A(;
      L     "RTE_405_DB".HMI.STEP_NUMBER;
      L     90;
      >=I;
      );
      =     "RTE_405_DB".FLAGS.STEP_END;

NETWORK
TITLE = COPY CURRENT STEP TO STEP TEXT WORD
      L     "RTE_405_DB".HMI.STEP_NUMBER;
      T     "RTE_405_DB".HMI.STEP_IDENT_TEXT_NUMBER;
      NOP   0;
END_FUNCTION
